(* Logix 5000 project; controller OptixWebinar 1756-L85E rev 35.11; software revision 35.00 *)

TASK MainTask (continuous, watchdog 500 ms) : MainProgram

MODULES
   Local : 1756-L85E (ICP 0, rev 35.11)
END_MODULES

TYPE UDT_SineWave :
STRUCT
   Offset : REAL;
   Frequency : REAL;
   Amplitude : REAL;
   Phase : REAL;
END_STRUCT
END_TYPE

ADD_ON_INSTRUCTION AOI_SineWave   (* revision 1.0, ExecutePrescan *)
VAR_IN_OUT
   Set : UDT_SineWave; {required}
END_VAR
VAR_OUTPUT
   Val_YValue : REAL; {access Read Only, visible}
END_VAR
VAR
   Wrk_ActualOffset : REAL;
   Wrk_OffsetDiff : REAL;
   Wrk_OffsetDiffABS : REAL;
   Wrk_1Percent : REAL;
   Wrk_LastCommandedSP : REAL;
   Wrk_10msTimer : TIMER := (PRE := 10);
   Wrk_TimeWindow : REAL;
   Wrk_Time_Generator : TIMER; {access None}
   Wrk_YValue : REAL;
   Wrk_ScratchPad2 : REAL;
   Wrk_ScratchPad1 : REAL;
   Wrk_Pi : REAL := 3.1416;
END_VAR

ROUTINE Logic   (* ladder *)
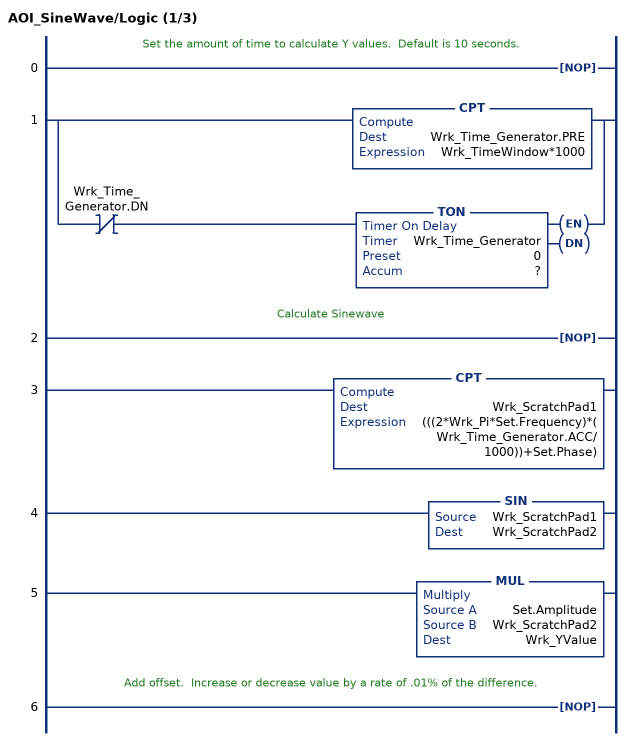
   // Set the amount of time to calculate Y values.  Default is 10 seconds.
   0: NOP();
   1: [CPT(Wrk_Time_Generator.PRE,Wrk_TimeWindow*1000) ,XIO(Wrk_Time_Generator.DN) TON(Wrk_Time_Generator,?,?) ];
   // Calculate Sinewave
   2: NOP();
   3: CPT(Wrk_ScratchPad1,(((2*Wrk_Pi*Set.Frequency)*(Wrk_Time_Generator.ACC/1000))+Set.Phase));
   4: SIN(Wrk_ScratchPad1,Wrk_ScratchPad2);
   5: MUL(Set.Amplitude,Wrk_ScratchPad2,Wrk_YValue);
   // Add offset.  Increase or decrease value by a rate of .01% of the difference.
   6: NOP();
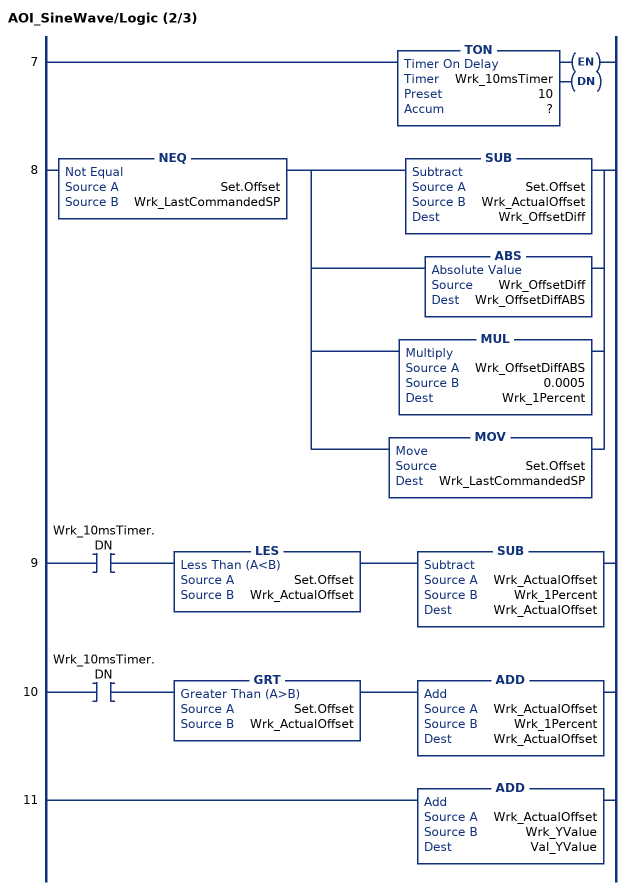
   7: TON(Wrk_10msTimer,?,?);
   8: NEQ(Set.Offset,Wrk_LastCommandedSP)[SUB(Set.Offset,Wrk_ActualOffset,Wrk_OffsetDiff) ,ABS(Wrk_OffsetDiff,Wrk_OffsetDiffABS) ,MUL(Wrk_OffsetDiffABS,0.0005,Wrk_1Percent) ,MOV(Set.Offset,Wrk_LastCommandedSP) ];
   9: XIC(Wrk_10msTimer.DN)LES(Set.Offset,Wrk_ActualOffset)SUB(Wrk_ActualOffset,Wrk_1Percent,Wrk_ActualOffset);
   10: XIC(Wrk_10msTimer.DN)GRT(Set.Offset,Wrk_ActualOffset)ADD(Wrk_ActualOffset,Wrk_1Percent,Wrk_ActualOffset);
   11: ADD(Wrk_ActualOffset,Wrk_YValue,Val_YValue);
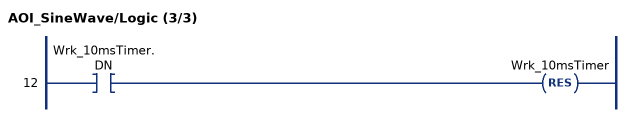
   12: XIC(Wrk_10msTimer.DN)RES(Wrk_10msTimer);
END_ROUTINE

ROUTINE Prescan   (* ladder *)
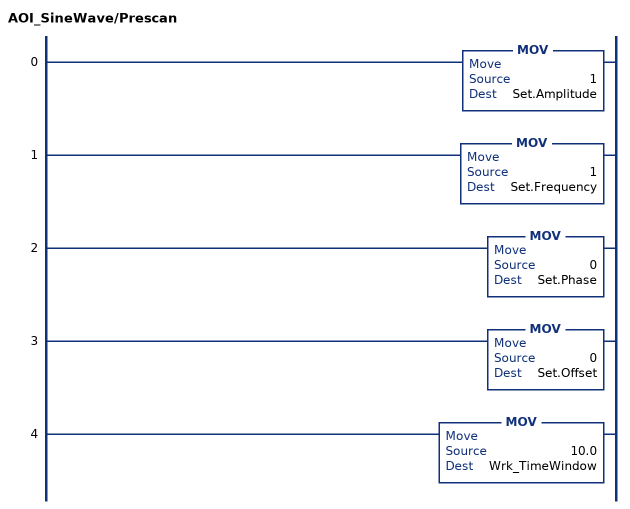
   0: MOV(1,Set.Amplitude);
   1: MOV(1,Set.Frequency);
   2: MOV(0,Set.Phase);
   3: MOV(0,Set.Offset);
   4: MOV(10.0,Wrk_TimeWindow);
END_ROUTINE
END_ADD_ON_INSTRUCTION

ADD_ON_INSTRUCTION Motor   (* revision 1.0 *)
VAR_INPUT
   OCmd_Start : BOOL;
   OCmd_Stop : BOOL;
END_VAR
VAR_OUTPUT
   Sts_Running : BOOL;
   Val_Speed : REAL;
END_VAR
VAR_INPUT
   OSet_SP : REAL;
END_VAR
VAR
   Wrk_SpeedSineWaveSettings : UDT_SineWave := (Frequency := 0.1, Amplitude := 0.2);
   Wrk_SpeedSineWave : AOI_SineWave;
END_VAR

ROUTINE Logic   (* ladder *)
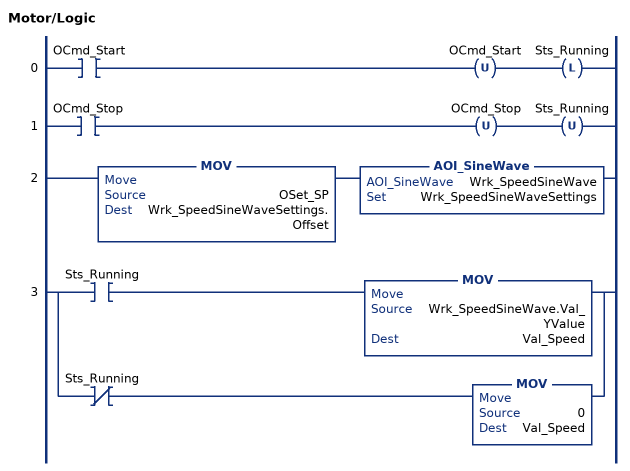
   0: XIC(OCmd_Start)OTU(OCmd_Start)OTL(Sts_Running);
   1: XIC(OCmd_Stop)OTU(OCmd_Stop)OTU(Sts_Running);
   2: MOV(OSet_SP,Wrk_SpeedSineWaveSettings.Offset)AOI_SineWave(Wrk_SpeedSineWave,Wrk_SpeedSineWaveSettings);
   3: [XIC(Sts_Running) MOV(Wrk_SpeedSineWave.Val_YValue,Val_Speed) ,XIO(Sts_Running) MOV(0,Val_Speed) ];
END_ROUTINE
END_ADD_ON_INSTRUCTION

VAR_GLOBAL   (* controller tags *)
   Motor1 : Motor := (Sts_Running := 1, Val_Speed := 20.102533, OSet_SP := 20.0);
   Motor2 : Motor := (Sts_Running := 1, Val_Speed := 45.23038, OSet_SP := 45.0);
   Motor3 : Motor := (Sts_Running := 1, Val_Speed := 50.309372, OSet_SP := 50.0);
END_VAR

PROGRAM MainProgram   (* main routine MainRoutine *)

ROUTINE MainRoutine   (* ladder *)
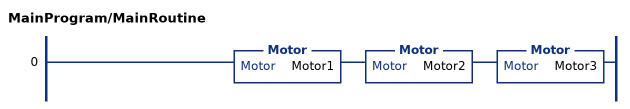
   0: Motor(Motor1)Motor(Motor2)Motor(Motor3);
END_ROUTINE
END_PROGRAM
